{attribute 'qualified_only'}
{attribute 'strict'}
// Sensor type: NO , NC
TYPE eSensorType :      
(
	NO := 0, 			// Normally opened
	NC       			// Normally closed
);
END_TYPE

(* stored: Version 1.1.0.1, ProductVersion 3.1.4024.12
   DUT eSensorType: Id {c739d113-6cf4-4eb4-82cd-5e0e9f7a42d1} *)
